# EPICS substitutions: mmcApp/Db/usbsn.substitutions
file usbsn.template
{
 pattern
 { BASE,          PORT,       SERIAL,        TIME          },
 { "\$(CTRL)",    "\$(ASYN)", "\$(SERIAL)",  "\$(TIME)",   }
}
